FUNCTION_BLOCK Wago1504_5 (* Service Interface Function Block Type *)
  (* Standard: 61499-2; Description: Copyright (c) 2018, 2024 fortiss GmbH This program and the accompanying materials are made available under the terms of the Eclipse Public License 2.0 which is available at https://www.eclipse.org/legal/epl-2.0/ SPDX-License-Identifier: EPL-2.0 *)
  (* Version 3.0, 2025-04-14, Patrick Aigner, changed package *)
  (* Version 1.1, 2024-09-22, Monika Wenger *)
  (* Version 1.0, 2018-12-05, Jose Cabral *)
  PACKAGE eclipse4diac::io::wago;
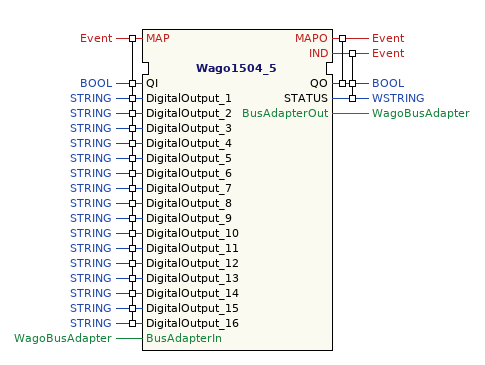
  EVENT_INPUT
    MAP WITH DigitalOutput_1, DigitalOutput_2, DigitalOutput_5, DigitalOutput_3, DigitalOutput_4, DigitalOutput_6, DigitalOutput_7, DigitalOutput_8, DigitalOutput_9, DigitalOutput_10, DigitalOutput_11, DigitalOutput_12, DigitalOutput_13, DigitalOutput_14, DigitalOutput_15, DigitalOutput_16, QI; (* Map Pins *)
  END_EVENT
  EVENT_OUTPUT
    MAPO WITH QO; (* Confirm Pin Mapping *)
    IND WITH QO, STATUS; (* Indication from Resource *)
  END_EVENT
  VAR_INPUT
    QI : BOOL; (* Event Input Qualifier *)
    DigitalOutput_1 : STRING;
    DigitalOutput_2 : STRING;
    DigitalOutput_3 : STRING;
    DigitalOutput_4 : STRING;
    DigitalOutput_5 : STRING;
    DigitalOutput_6 : STRING;
    DigitalOutput_7 : STRING;
    DigitalOutput_8 : STRING;
    DigitalOutput_9 : STRING;
    DigitalOutput_10 : STRING;
    DigitalOutput_11 : STRING;
    DigitalOutput_12 : STRING;
    DigitalOutput_13 : STRING;
    DigitalOutput_14 : STRING;
    DigitalOutput_15 : STRING;
    DigitalOutput_16 : STRING;
  END_VAR
  VAR_OUTPUT
    QO : BOOL; (* Event Output Qualifier *)
    STATUS : WSTRING; (* Service Status *)
  END_VAR
  SOCKETS
    BusAdapterIn : eclipse4diac::io::wago::WagoBusAdapter;
  END_SOCKETS
  PLUGS
    BusAdapterOut : eclipse4diac::io::wago::WagoBusAdapter;
  END_PLUGS
END_FUNCTION_BLOCK
